// TIA Portal V16 export
// export: Created 2021-11-12T13:31:34.3086039Z, ExportSetting WithDefaults, DisplayName Totally Integrated Automation Portal, DisplayVersion V16 Update 3, DisplayName TIA Portal Version Control Interface, DisplayVersion V16 Update 2, DisplayName TIA Portal Openness, DisplayVersion V16 Update 3, DisplayName SINAMICS Startdrive Advanced, DisplayVersion V16 Update 5, DisplayName SINAMICS Startdrive G130, G150, S120, S150, SINAMICS MV, S210, DisplayVersion V16 Update 5, DisplayName SINAMICS Startdrive G110M, G120, G120C, G120D, G120P, G115D, DisplayVersion V16 Update 5, DisplayName STEP 7 Professional, DisplayVersion V16 Update 3, DisplayName STEP 7 Safety, DisplayVersion V16, DisplayName WinCC UA Professional, DisplayVersion V16 Update 3
FUNCTION_BLOCK "TrackLubrication"   // FB23, LAD
{ S7_Optimized_Access := 'TRUE' }
VERSION : 0.1
// stored: AutoNumber true, IsIECCheckEnabled false, IsRetainMemResEnabled false, MemoryReserve 100, SetENOAutomatically false, UDAEnableTagReadback false
   VAR_INPUT
      IS_ZoneM { ExternalAccessible := 'False'; ExternalVisible := 'False'; ExternalWritable := 'False'} : "UDT_Status_main";   // Main structure from zone
      IS_ZoneS { ExternalAccessible := 'False'; ExternalVisible := 'False'; ExternalWritable := 'False'} : "UDT_Zone_Status_specific";   // Specific structure from zone
      IB1Senzor : Bool;   // Lubrication printed feedback
      II_NoOfCycles : Int;   // Number of cycles to lubricate if no feedback from senzor
      IT_Interval : Time;   // Interval to repeat lubrication
      IT_Lubricate : Time;   // Duration of lubrication
      IT_Break : Time;   // Duration of breake between cycles
      IT_OnDel : Time;   // TON filtration
   END_VAR
   VAR_OUTPUT
      OB1Pump : Bool;   // Start pump
      OB1Error : Bool;   // Tank empty, senzor error, pump error
   END_VAR
   VAR
      ST_TONLubricate { S7_SetPoint := 'True'} : TON_TIME;
      ST_TPLubricate { S7_SetPoint := 'True'} : TP_TIME;
      ST_TPBreak { S7_SetPoint := 'True'} : TON_TIME;
      ST_TONFilter { S7_SetPoint := 'True'} : TON_TIME;
      ST_TONFilter_1 { S7_SetPoint := 'True'} : TON_TIME;
      ST_Counter { S7_SetPoint := 'True'} : CTU_INT;   // Number of unnsuccessfull cycles
   END_VAR
   VAR RETAIN
      SB1LubricOk : Bool;   // Lubrication successful
      SB1LubricNok : Bool;   // Lubrication not successful
   END_VAR
   VAR
      SB1Break : Bool;   // Break between cycles
      SB1LubricInProcess : Bool;   // Lubrication process running
   END_VAR
   VAR_TEMP
      TB1Error : Bool;
   END_VAR
BEGIN

REGION Network 1: Clear temporary variables
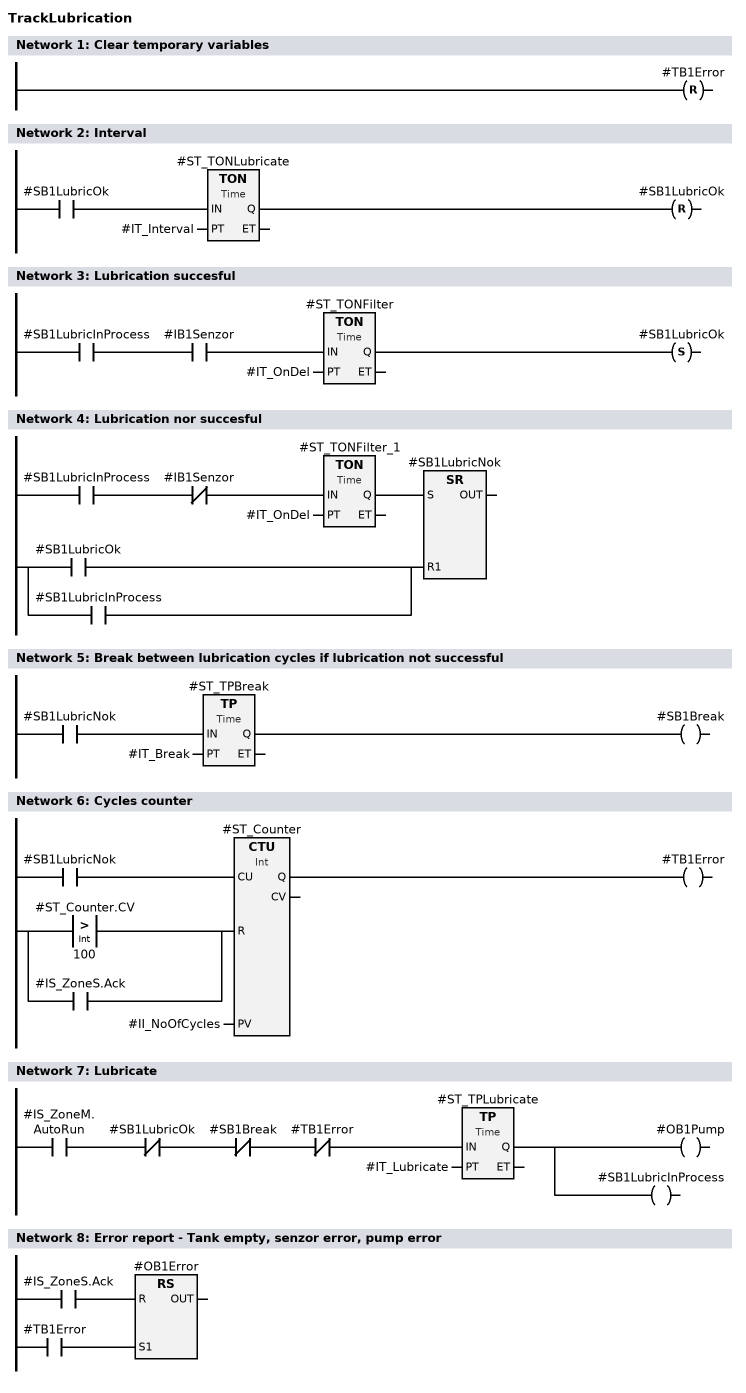
   RUNG wire#powerrail
      R_Coil( #TB1Error )
   END_RUNG
   // the same network as SCL:
   #TB1Error := FALSE;
END_REGION

REGION Network 2: Interval
   RUNG wire#powerrail
      Contact( #SB1LubricOk )
      { S7_Templates := "time_type := Time" } #ST_TONLubricate.TON(pt := #IT_Interval, et =>)
      R_Coil( #SB1LubricOk )
   END_RUNG
   // the same network as SCL:
   #ST_TONLubricate(IN := #SB1LubricOk, PT := #IT_Interval);   // TON
   IF #ST_TONLubricate.Q THEN #SB1LubricOk := FALSE; END_IF;
END_REGION

REGION Network 3: Lubrication succesful
   RUNG wire#powerrail
      Contact( #SB1LubricInProcess )
      Contact( #IB1Senzor )
      { S7_Templates := "time_type := Time" } #ST_TONFilter.TON(pt := #IT_OnDel, et =>)
      S_Coil( #SB1LubricOk )
   END_RUNG
   // the same network as SCL:
   #ST_TONFilter(IN := #SB1LubricInProcess AND #IB1Senzor, PT := #IT_OnDel);   // TON
   IF #ST_TONFilter.Q THEN #SB1LubricOk := TRUE; END_IF;
END_REGION

REGION Network 4: Lubrication nor succesful
   RUNG wire#powerrail
      Contact( #SB1LubricInProcess )
      I_Contact( #IB1Senzor )
      { S7_Templates := "time_type := Time" } #ST_TONFilter_1.TON(pt := #IT_OnDel, et =>)
      S_SR(operand := #SB1LubricNok, r1 := wire#w1)
   END_RUNG
   RUNG wire#powerrail
      Contact( #SB1LubricOk )
   END_RUNG wire#w1
   RUNG wire#powerrail
      Contact( #SB1LubricInProcess )
   END_RUNG wire#w1
   // the same network as SCL:
   #ST_TONFilter_1(IN := #SB1LubricInProcess AND NOT #IB1Senzor, PT := #IT_OnDel);   // TON
   IF #ST_TONFilter_1.Q THEN
       #SB1LubricNok := TRUE;   // SR flip-flop
   END_IF;
   IF #SB1LubricOk OR #SB1LubricInProcess THEN #SB1LubricNok := FALSE; END_IF;
END_REGION

REGION Network 5: Break between lubrication cycles if lubrication not successful
   RUNG wire#powerrail
      Contact( #SB1LubricNok )
      { S7_Templates := "time_type := Time" } #ST_TPBreak.TP(pt := #IT_Break, et =>)
      Coil( #SB1Break )
   END_RUNG
   // the same network as SCL:
   #ST_TPBreak(IN := #SB1LubricNok, PT := #IT_Break);   // TP
   #SB1Break := #ST_TPBreak.Q;
END_REGION

REGION Network 6: Cycles counter
   RUNG wire#powerrail
      Contact( #SB1LubricNok )
      { S7_Templates := "value_type := Int" } #ST_Counter.CTU(r := wire#w1, pv := #II_NoOfCycles, cv =>)
      Coil( #TB1Error )
   END_RUNG
   RUNG wire#powerrail
      { S7_Templates := "SrcType := Int" } GT_Contact(in1 := #ST_Counter.CV, in2 := 100)
   END_RUNG wire#w1
   RUNG wire#powerrail
      Contact( #IS_ZoneS.Ack )
   END_RUNG wire#w1
   // the same network as SCL:
   #ST_Counter(CU := #SB1LubricNok, R := (#ST_Counter.CV > 100) OR #IS_ZoneS.Ack, PV := #II_NoOfCycles);   // CTU
   #TB1Error := #ST_Counter.Q;
END_REGION

REGION Network 7: Lubricate
   RUNG wire#powerrail
      Contact( #IS_ZoneM.AutoRun )
      I_Contact( #SB1LubricOk )
      I_Contact( #SB1Break )
      I_Contact( #TB1Error )
      { S7_Templates := "time_type := Time" } #ST_TPLubricate.TP(pt := #IT_Lubricate, et =>)
      wire#w1
      Coil( #OB1Pump )
   END_RUNG
   RUNG wire#w1
      Coil( #SB1LubricInProcess )
   END_RUNG
   // the same network as SCL:
   #ST_TPLubricate(IN := #IS_ZoneM.AutoRun AND NOT #SB1LubricOk AND NOT #SB1Break AND NOT #TB1Error,   // TP
                   PT := #IT_Lubricate);
   #OB1Pump := #ST_TPLubricate.Q;
   #SB1LubricInProcess := #ST_TPLubricate.Q;
END_REGION

REGION Network 8: Error report - Tank empty, senzor error, pump error
   RUNG wire#powerrail
      Contact( #IS_ZoneS.Ack )
      S_RS(operand := #OB1Error, s1 := wire#w1)
   END_RUNG
   RUNG wire#powerrail
      Contact( #TB1Error )
   END_RUNG wire#w1
   // the same network as SCL:
   IF #IS_ZoneS.Ack THEN
       #OB1Error := FALSE;   // RS flip-flop
   END_IF;
   IF #TB1Error THEN #OB1Error := TRUE; END_IF;
END_REGION
END_FUNCTION_BLOCK
